Yaskawa INFORM job: TRIANGU.JBI

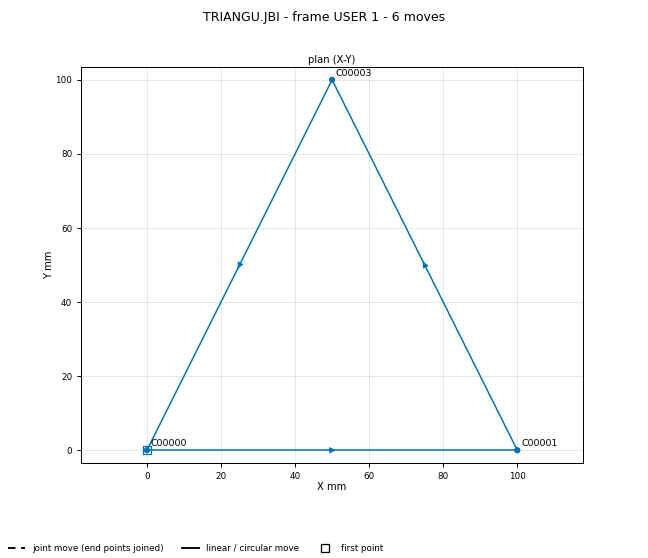
[picture p0: tool path of TRIANGU.JBI in frame USER 1, 6 of 6 moves have a stored position in this frame; points joined in program order, loops and branches not executed]
/JOB
//NAME TRIANGU
//POS
///NPOS 6,0,0,0,0,0
///USER 1
///TOOL 1
///POSTYPE USER
///RECTAN
///RCONF 1,0,0,0,0,0,0,0,0,0,0,0,0,0,0,0,0,0,0,0,0,0,0,0
C00000=0.000,0.000,7.000,0.0000,0.0000,0.0000
C00001=100.000,0.000,7.000,0.0000,0.0000,0.0000
C00002=100.000,0.000,7.000,0.0000,0.0000,0.0000
C00003=50.000,100.000,7.000,0.0000,0.0000,0.0000
C00004=50.000,100.000,7.000,0.0000,0.0000,0.0000
C00005=0.000,0.000,7.000,0.0000,0.0000,0.0000
//INST
///DATE 2025/05/20 16:00
///ATTR SC,RW,RJ
////FRAME USER 1
///GROUP1 RB1
NOP
MOVJ C00000 VJ=30.00
DOUT OT#(1) ON
TIMER T=1.000
MOVL C00001 V=40.0 PL=0
DOUT OT#(1) OFF
TIMER T=1.000
MOVJ C00002 VJ=30.00
DOUT OT#(1) ON
TIMER T=1.000
MOVL C00003 V=40.0 PL=0
DOUT OT#(1) OFF
TIMER T=1.000
MOVJ C00004 VJ=30.00
DOUT OT#(1) ON
TIMER T=1.000
MOVL C00005 V=40.0 PL=0
DOUT OT#(1) OFF
TIMER T=1.000
END
